{attribute 'GeneratedUsingTerminal: KL9210'}
{attribute addProperty BoxType "KL9210"}
{attribute addProperty Id "Channel_1AT %I*Channel_64AAC8C70"}
{attribute addProperty CRC "2347652594"}
{attribute addProperty Size "0"}
TYPE KL9210_8BEE55F2 :
STRUCT
	{attribute addProperty Name "Channel_1"}
	Channel_1 : Channel_64AAC8C7;
END_STRUCT
END_TYPE

(* stored: Version 1.2.0.0, ProductVersion 3.1.4024.9
   DUT KL9210_8BEE55F2: Id {e3e1b1d8-6bb4-413e-ba48-c594df4d758a} *)
